{attribute 'qualified_only'}
VAR_GLOBAL PERSISTENT
	AirKnife_VFD : VFD;
	AirKnife_Start : BOOL;
	AirKnife_Percent_Speed_Input : REAL := 100;
	AirKnife_StartwithSystem : BOOL;
	AirKnife_Analog_Input AT %I* : INT;
	AirKnife_Filter_Change_Setting : REAL := 15;
	AirKnife_Vacuum_Level : REAL;
END_VAR

(* stored: Version 1.1.0.1, ProductVersion 3.1.4024.12
   GVL GVL_AirKnife: Id {fba7f8c3-ca7c-4ca1-9410-ab9c3820f962} *)
